INTERFACE I_Observer EXTENDS __SYSTEM.IQueryInterface

PROPERTY nTypeClass : __SYSTEM.TYPE_CLASS
GET
END_GET
END_PROPERTY

METHOD Update : I_Observer
VAR_INPUT
    anyVal:         ANY;
END_VAR
END_METHOD

END_INTERFACE

(* stored: Version 1.1.0.1, ProductVersion 3.1.4024.12
   Itf I_Observer: Id {71e9c537-c1c0-4a93-aa9e-3a7f11d757ab}
   Property nTypeClass: Id {45bcd299-a5df-005e-250a-29bf5493035a}
   Get Get: Id {abae06e7-3ed9-0451-2c99-f3ae104e17eb}
   Method Update: Id {fcb17013-ca2e-40da-951a-a3620cf618d3} *)
